
FUNCTION CB_int_to_dint : DINT

TITLE = ' Convert an integer into a Dint '
VERSION : '1.0'
AUTHOR  : CB
NAME    : intToDin
FAMILY  : TNI

VAR_INPUT
    IN : INT;
END_VAR

BEGIN

CB_int_to_dint := INT_TO_DINT(IN);

END_FUNCTION
